TYPE ST_CommunicatorMassege :
STRUCT
	sText				: STRING;
	bToPickUp			: BOOL;		//informacja ze komunikat jest aktualny, po odebraniu przez odbiorce flaga znika
	bValue				: BOOL;
	rValue				: REAL;
END_STRUCT
END_TYPE

(* stored: Version 1.1.0.1
   DUT ST_CommunicatorMassege: Id {d2956b33-e0a3-00fe-217d-27d07a890ff6} *)
